% RSLogix 500 project I2P JOB 14 - MYAH.RSS, saved by version 10.00.00.00 %
PROJECT "ML05B"    % processor: Bul.1763 MicroLogix 1100 Series B %

PROGRAM FILES
  LAD 2   13 rungs

DATA FILES
  O0 OUTPUT  4 elements
  I1 INPUT  6 elements
  S2 STATUS  66 elements
  B3 BINARY  1 elements
  T4 TIMER  1 elements
  C5 COUNTER  1 elements
  R6 CONTROL  1 elements
  N7 INTEGER  1 elements
  F8 FLOAT  1 elements

LADDER 2
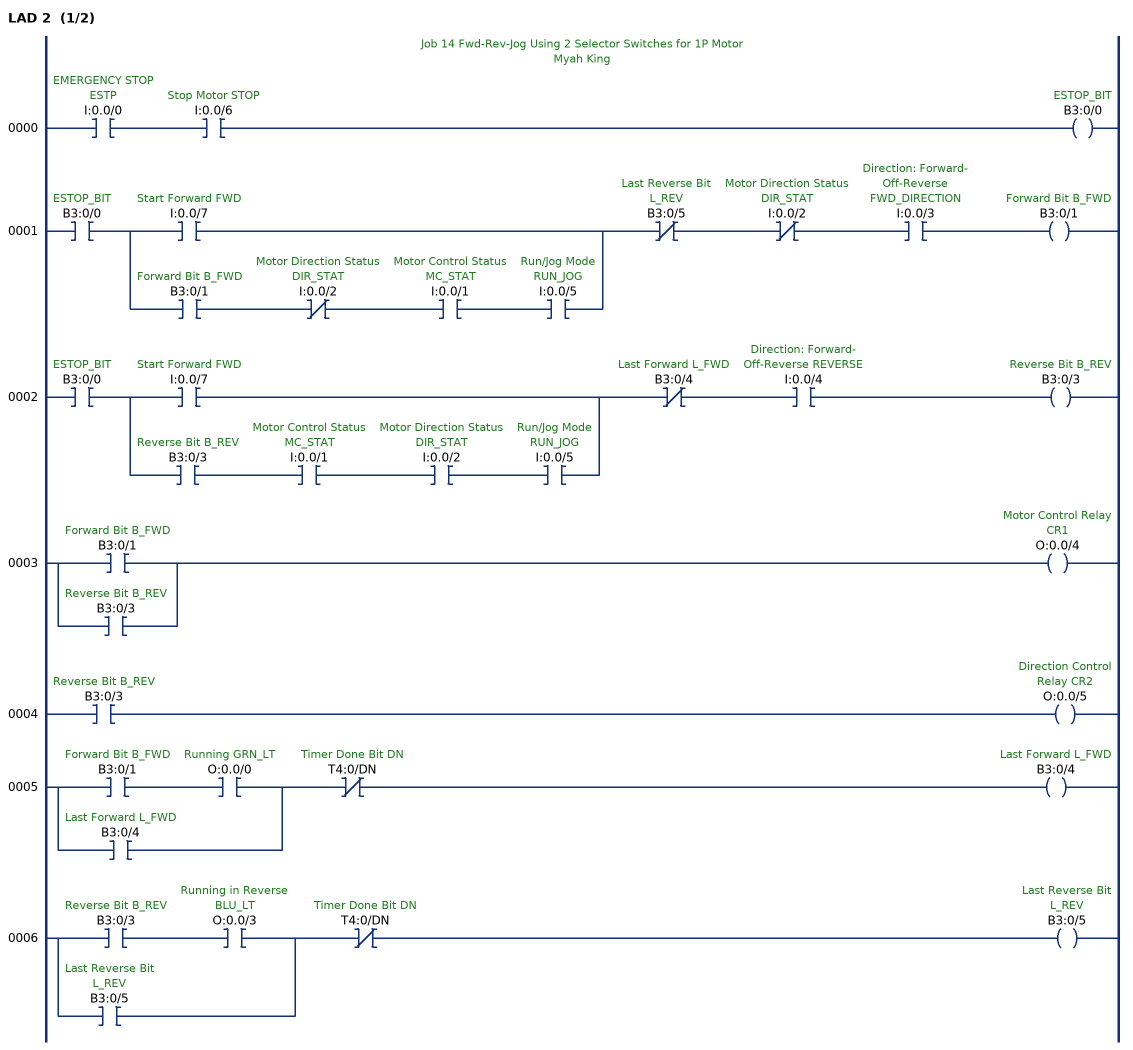
% Rung: 0 %
% Job 14 Fwd-Rev-Jog Using 2 Selector Switches for 1P Motor
% Myah King %
SOR XIC I:0.0/0 XIC I:0.0/6 OTE B3:0/0 EOR
%   I:0.0/0  ESTP  "EMERGENCY STOP" %
%   I:0.0/6  STOP  "Stop Motor" %
%   B3:0/0  ESTOP_BIT %
% Rung: 1 %
SOR XIC B3:0/0 BST XIC I:0.0/7 NXB XIC B3:0/1 XIO I:0.0/2 XIC I:0.0/1 XIC I:0.0/5 BND XIO B3:0/5 XIO I:0.0/2 XIC I:0.0/3 OTE B3:0/1 EOR
%   B3:0/0  ESTOP_BIT %
%   I:0.0/7  FWD  "Start Forward" %
%   B3:0/1  B_FWD  "Forward Bit" %
%   I:0.0/2  DIR_STAT  "Motor Direction Status" %
%   I:0.0/1  MC_STAT  "Motor Control Status" %
%   I:0.0/5  RUN_JOG  "Run/Jog Mode" %
%   B3:0/5  L_REV  "Last Reverse Bit" %
%   I:0.0/3  FWD_DIRECTION  "Direction: Forward- Off-Reverse" %
% Rung: 2 %
SOR XIC B3:0/0 BST XIC I:0.0/7 NXB XIC B3:0/3 XIC I:0.0/1 XIC I:0.0/2 XIC I:0.0/5 BND XIO B3:0/4 XIC I:0.0/4 OTE B3:0/3 EOR
%   B3:0/0  ESTOP_BIT %
%   I:0.0/7  FWD  "Start Forward" %
%   B3:0/3  B_REV  "Reverse Bit" %
%   I:0.0/1  MC_STAT  "Motor Control Status" %
%   I:0.0/2  DIR_STAT  "Motor Direction Status" %
%   I:0.0/5  RUN_JOG  "Run/Jog Mode" %
%   B3:0/4  L_FWD  "Last Forward" %
%   I:0.0/4  REVERSE  "Direction: Forward- Off-Reverse" %
% Rung: 3 %
SOR BST XIC B3:0/1 NXB XIC B3:0/3 BND OTE O:0.0/4 EOR
%   B3:0/1  B_FWD  "Forward Bit" %
%   B3:0/3  B_REV  "Reverse Bit" %
%   O:0.0/4  CR1  "Motor Control Relay" %
% Rung: 4 %
SOR XIC B3:0/3 OTE O:0.0/5 EOR
%   B3:0/3  B_REV  "Reverse Bit" %
%   O:0.0/5  CR2  "Direction Control Relay" %
% Rung: 5 %
SOR BST XIC B3:0/1 XIC O:0.0/0 NXB XIC B3:0/4 BND XIO T4:0/DN OTE B3:0/4 EOR
%   B3:0/1  B_FWD  "Forward Bit" %
%   O:0.0/0  GRN_LT  "Running" %
%   B3:0/4  L_FWD  "Last Forward" %
%   T4:0/DN  DN  "Timer Done Bit" %
% Rung: 6 %
SOR BST XIC B3:0/3 XIC O:0.0/3 NXB XIC B3:0/5 BND XIO T4:0/DN OTE B3:0/5 EOR
%   B3:0/3  B_REV  "Reverse Bit" %
%   O:0.0/3  BLU_LT  "Running in Reverse" %
%   B3:0/5  L_REV  "Last Reverse Bit" %
%   T4:0/DN  DN  "Timer Done Bit" %

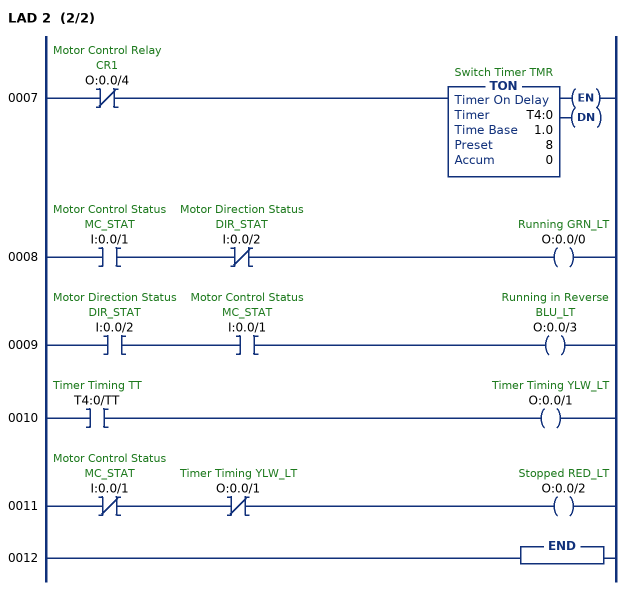
% Rung: 7 %
SOR XIO O:0.0/4 TON T4:0 1.0 8 0 EOR
%   O:0.0/4  CR1  "Motor Control Relay" %
%   T4:0  TMR  "Switch Timer" %
% Rung: 8 %
SOR XIC I:0.0/1 XIO I:0.0/2 OTE O:0.0/0 EOR
%   I:0.0/1  MC_STAT  "Motor Control Status" %
%   I:0.0/2  DIR_STAT  "Motor Direction Status" %
%   O:0.0/0  GRN_LT  "Running" %
% Rung: 9 %
SOR XIC I:0.0/2 XIC I:0.0/1 OTE O:0.0/3 EOR
%   I:0.0/2  DIR_STAT  "Motor Direction Status" %
%   I:0.0/1  MC_STAT  "Motor Control Status" %
%   O:0.0/3  BLU_LT  "Running in Reverse" %
% Rung: 10 %
SOR XIC T4:0/TT OTE O:0.0/1 EOR
%   T4:0/TT  TT  "Timer Timing" %
%   O:0.0/1  YLW_LT  "Timer Timing" %
% Rung: 11 %
SOR XIO I:0.0/1 XIO O:0.0/1 OTE O:0.0/2 EOR
%   I:0.0/1  MC_STAT  "Motor Control Status" %
%   O:0.0/1  YLW_LT  "Timer Timing" %
%   O:0.0/2  RED_LT  "Stopped" %
% Rung: 12 %
SOR END EOR

OTHER DOCUMENTED ADDRESSES
  I:0.0/8  REV  "Start Reverse"

DATA TABLE (non-zero values as saved)
DATA B3
% B3:0 % 0X0001
DATA T4
% .PRE .ACC %
% T4:0 % 8 0
